// TIA Portal V19 export
FUNCTION "Conv_BOOL_to_STRING" : String   // FC90, LAD
// stored: Access Published, SetENOAutomatically false
   VAR_INPUT
      BooleanValue : Bool;
      sType : UInt;   // Stringhe per conversione valore booleano: 0= TRUE/FALSE; 1= ON/OFF
   END_VAR
BEGIN

REGION Network 1 (SCL): BOOL -> STRING
   IF #BooleanValue THEN

       CASE #sType OF
           1:
               #Conv_BOOL_to_STRING := 'ON';
           ELSE
               #Conv_BOOL_to_STRING := 'TRUE';
       END_CASE;




   ELSE
       CASE #sType OF
           1:
               #Conv_BOOL_to_STRING := 'OFF';
           ELSE
               #Conv_BOOL_to_STRING := 'FALSE';
       END_CASE;



   END_IF;
END_REGION
END_FUNCTION
